// TIA Portal V20 export
// export: Created 2025-12-01T14:57:06.3862051Z, ExportSetting None, DisplayName Totally Integrated Automation Portal, DisplayVersion V20 Update 3, DisplayName TIA Portal Openness, DisplayVersion V20 Update 3, DisplayName TIA Portal Version Control Interface, DisplayVersion V20 Update 3, DisplayName STEP 7 Professional, DisplayVersion V20 Update 3, DisplayName STEP 7 Safety, DisplayVersion V20 Update 2, DisplayName WinCC Basic/Comfort/Advanced, DisplayVersion V20 Update 3, DisplayName WinCC Professional, DisplayVersion V20 Update 3, DisplayName WinCC Unified, DisplayVersion V20 Update 3
FUNCTION "FC978_PosiControl_VarLenze" : Void   // FC978, LAD
{ S7_Optimized_Access := 'FALSE' }
// stored: AutoNumber false, SetENOAutomatically false
   VAR_INPUT
      Estado_CB : "EstadoZona";
      Error_Tx : Bool;
      NodoNoPresente : Bool;
      ByteInicial : Int;
      Velocidad_FR : Int;
      MaxVelocidad_FR : Int;
      EM_Up : Bool;
      EM_Dw : Bool;
      pHsProtusion : Bool;
      SubirManual : Bool;
      BajarManual : Bool;
      Homing : Bool;
      ModoHormingAuto : Bool;
      pHsReferencia : Bool;
      Orden : Bool;
      PosicionOrden : Int;
   END_VAR
   VAR_OUTPUT
      Error_SubjetArea : Word;
      Error_IDArea : Word;
      FinOrden : Bool;
   END_VAR
   VAR_IN_OUT
      PosicionActual : Int;
      ReferenciaOK : Bool;
      ErrorVariador : Bool;
      MemoHomingAuto : Bool;
   END_VAR
   VAR_TEMP
      InVar : Struct
         EnPosicion : Bool;   // Indica que el variador esta posicionado dentro de unos margenes
         EnMovimiento : Bool;   // Indica que el variador esta realizando una orden
         ReferenciaOK : Bool;   // Indica que el variador esta bien referenciado desde la posicion de origen
         HomingDone : Bool;
         SelecMotor_Bit1 : Bool;
         SelecMotor_Bit2 : Bool;
         Libre_Bit14 : Bool;
         Libre_Bit15 : Bool;
         Error_Var : Bool;   // Esto nos indica que hay un erro en el variador
         Libre_Bit1 : Bool;
         Libre_Bit2 : Bool;
         Inhivido : Bool;   // Señal Inhivir var actibo
         Ready_Var : Bool;   // Nos indica que el variador esta listo para realizar los movimientos
         Libre_Bit5 : Bool;
         Libre_Bit6 : Bool;
         Welltime : Bool;
      END_STRUCT;
      OutVar : Struct
         Ejecutar_Posicionamiento : Bool;   // Se activa para dar marcha
         EnableSpeedOveride : Bool;   // Para habilitar el speedoveride
         Reset_Homing : Bool;   // Para referenciar de nuevo el elevador
         Rearme_Var : Bool;
         Set_Homing : Bool;
         pHsReferencia : Bool;
         Manual_Subir : Bool;
         Manual_Bajar : Bool;
         Libre_Bit0 : Bool;
         Libre_Bit1 : Bool;
         Libre_Bit2 : Bool;
         Inhivir_Variador : Bool;   // Señal para inhivir el variador
         Modo_Homming : Bool;   // Tiene que estar activado para refernciar el elevador a cero
         Modo_Manual : Bool;   // Tiene que estar a uno para hacer movimiento en manual
         Modo_AutoRemoto : Bool;   // Tiene que estar a uno para lanzar el posicionamiento
         Libre_Bit7 : Bool;
      END_STRUCT;
      SpeedOrverride : Int;
      P_InVar : DWord;
      P_OutVar : DWord;
      PosicionDestino : Int;
      P_ByteInicialVar : DWord;
      P_Temporal : DWord;
      TempVelocidad : DInt;
      TempVelocidadMax : DInt;
      Margen : Int;
      PosDestinoMinimo : Int;
      PosDestinoMaximo : Int;
   END_VAR
BEGIN

REGION Network 1: Inicializacion
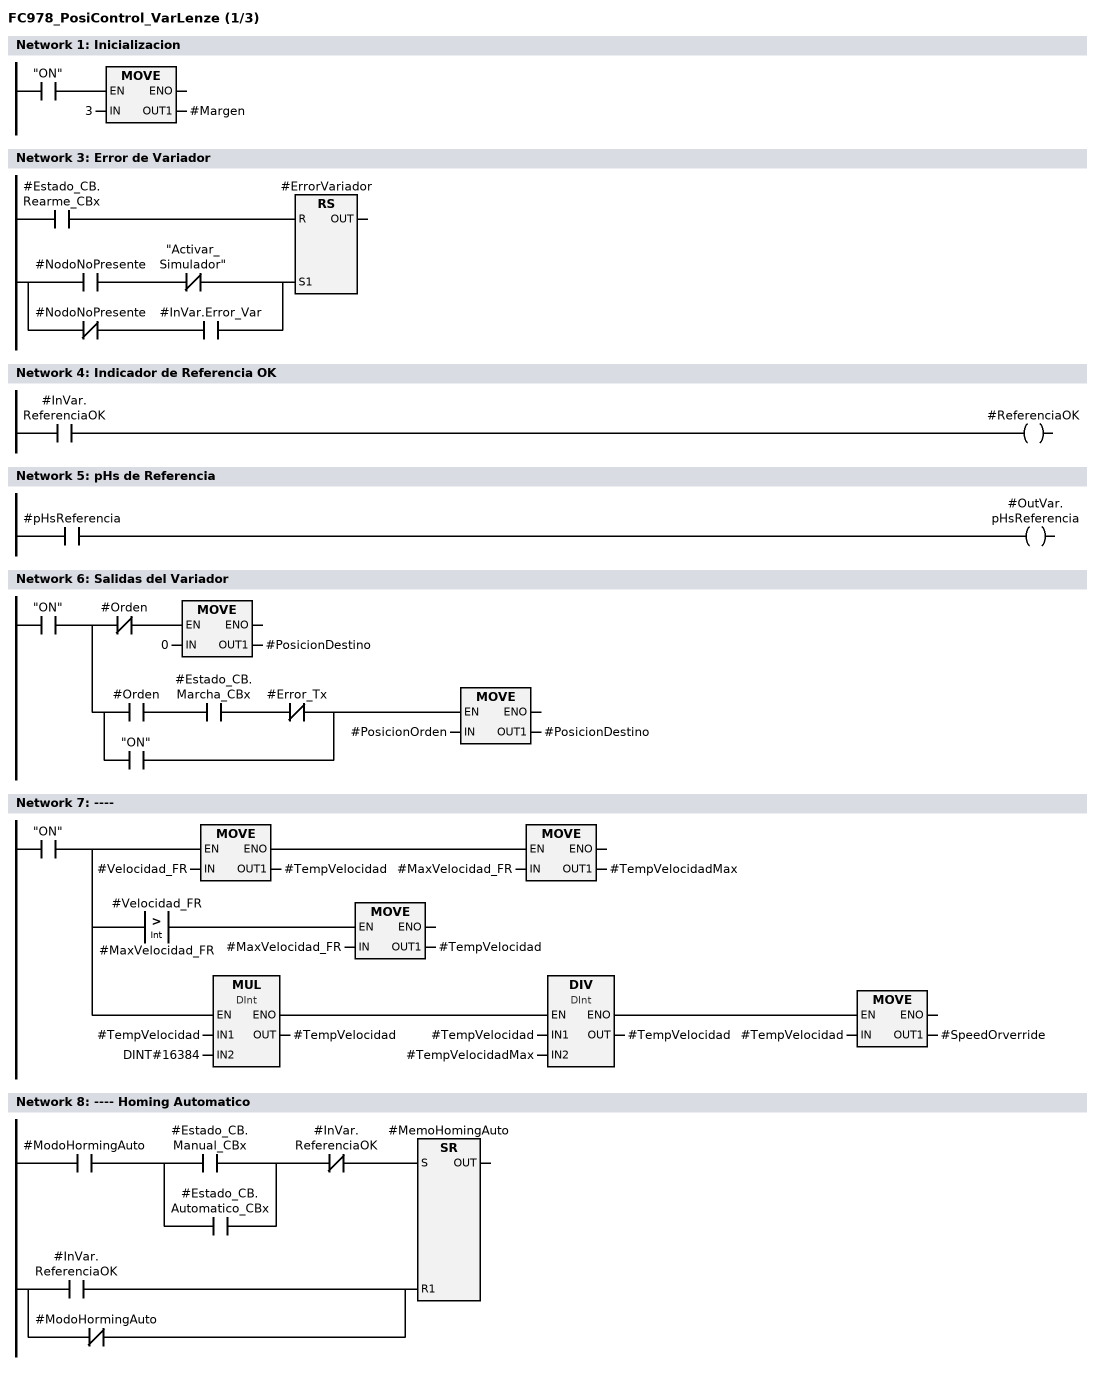
   RUNG wire#powerrail
      Contact( "ON" )
      { S7_GenerateENO := "TRUE" } Move(in := 3, out1 => #Margen)
   END_RUNG
   // the same network as SCL:
   IF "ON" THEN #Margen := 3; END_IF;
END_REGION

NETWORK
TITLE = Lectura del Variador
// -------------------------------------------------------------------
// --- Inicializar las Variables Internas

      L     P##InVar;  // Punteros a las variables internas
      T     #P_InVar;
      L     P##OutVar;
      T     #P_OutVar;

      L     #ByteInicial;  // Puntero al Variador
      SLD   3;
      T     #P_ByteInicialVar;

      L     0;  // Inicializar las variables internas
      T     LW [#P_InVar];
      T     LW [#P_OutVar];

      A     #NodoNoPresente;
      JC    NoLecturaVariador;

// -------------------------------------------------------------------
// --- Lectura de Datos del Variador

      L     #P_ByteInicialVar;  // Leer el Word p#0.0 del Variador
      L     P#0.0;  // Status del Variador "IN"
      +D;
      T     #P_Temporal;

      L     IW [#P_Temporal];
      T     LW [#P_InVar];

      L     #P_ByteInicialVar;  // Leer el Word p#2.0 del Variador
      L     P#2.0;  // Posicion Actual
      +D;
      T     #P_Temporal;

      L     IW [#P_Temporal];
      T     #PosicionActual;

// --- Codigo de Error

      L     #P_ByteInicialVar;  // Leer el Word p#6.0 del Variador
      L     P#6.0;  // ID Area del Variador
      +D;
      T     #P_Temporal;

      L     IW [#P_Temporal];
      T     #Error_IDArea;

      L     #P_ByteInicialVar;  // Leer el Word p#8.0 del Variador
      L     P#8.0;  // Subject Area del Variador
      +D;
      T     #P_Temporal;

      L     IW [#P_Temporal];
      T     #Error_SubjetArea;

// -------------------------------------------------------------------
// --- Final de Lectura de Datos del Variados

NoLecturaVariador:NOP   0;


REGION Network 3: Error de Variador
   RUNG wire#powerrail
      Contact( #Estado_CB.Rearme_CBx )
      S_RS(operand := #ErrorVariador, s1 := wire#w1)
   END_RUNG
   RUNG wire#powerrail
      Contact( #NodoNoPresente )
      I_Contact( "Activar_Simulador" )
   END_RUNG wire#w1
   RUNG wire#powerrail
      I_Contact( #NodoNoPresente )
      Contact( #InVar.Error_Var )
   END_RUNG wire#w1
   // the same network as SCL:
   IF #Estado_CB.Rearme_CBx THEN
       #ErrorVariador := FALSE;   // RS flip-flop
   END_IF;
   IF (#NodoNoPresente AND NOT "Activar_Simulador") OR (NOT #NodoNoPresente AND #InVar.Error_Var) THEN
       #ErrorVariador := TRUE;
   END_IF;
END_REGION

REGION Network 4: Indicador de Referencia OK
   RUNG wire#powerrail
      Contact( #InVar.ReferenciaOK )
      Coil( #ReferenciaOK )
   END_RUNG
   // the same network as SCL:
   #ReferenciaOK := #InVar.ReferenciaOK;
END_REGION

REGION Network 5: pHs de Referencia
   RUNG wire#powerrail
      Contact( #pHsReferencia )
      Coil( #OutVar.pHsReferencia )
   END_RUNG
   // the same network as SCL:
   #OutVar.pHsReferencia := #pHsReferencia;
END_REGION

REGION Network 6: Salidas del Variador
   RUNG wire#powerrail
      Contact( "ON" )
      wire#w1
      I_Contact( #Orden )
      { S7_GenerateENO := "TRUE" } Move(in := 0, out1 => #PosicionDestino)
   END_RUNG
   RUNG wire#w1
      Contact( #Orden )
      Contact( #Estado_CB.Marcha_CBx )
      I_Contact( #Error_Tx )
      wire#w2
      { S7_GenerateENO := "TRUE" } Move(in := #PosicionOrden, out1 => #PosicionDestino)
   END_RUNG
   RUNG wire#w1
      Contact( "ON" )
   END_RUNG wire#w2
   // the same network as SCL:
   IF "ON" AND NOT #Orden THEN #PosicionDestino := 0; END_IF;
   IF "ON" AND ((#Orden AND #Estado_CB.Marcha_CBx AND NOT #Error_Tx) OR "ON") THEN
       #PosicionDestino := #PosicionOrden;
   END_IF;
END_REGION

REGION Network 7: ----
   RUNG wire#powerrail
      Contact( "ON" )
      wire#w1
      { S7_GenerateENO := "TRUE" } Move(in := #Velocidad_FR, out1 => #TempVelocidad)
      { S7_GenerateENO := "TRUE" } Move(in := #MaxVelocidad_FR, out1 => #TempVelocidadMax)
   END_RUNG
   RUNG wire#w1
      { S7_Templates := "SrcType := Int" } GT_Contact(in1 := #Velocidad_FR, in2 := #MaxVelocidad_FR)
      { S7_GenerateENO := "TRUE" } Move(in := #MaxVelocidad_FR, out1 => #TempVelocidad)
   END_RUNG
   RUNG wire#w1
      { S7_Templates := "SrcType := DInt"; S7_GenerateENO := "TRUE" } Mul(in1 := #TempVelocidad, in2 := DINT#16384, out => #TempVelocidad)
      { S7_Templates := "SrcType := DInt"; S7_GenerateENO := "TRUE" } Div(in1 := #TempVelocidad, in2 := #TempVelocidadMax, out => #TempVelocidad)
      { S7_GenerateENO := "TRUE" } Move(in := #TempVelocidad, out1 => #SpeedOrverride)
   END_RUNG
   // the same network as SCL:
   // ENO of a box is taken as its EN; it also drops when the box reports an error
   IF "ON" THEN
       #TempVelocidad := #Velocidad_FR;
       #TempVelocidadMax := #MaxVelocidad_FR;
   END_IF;
   IF "ON" AND (#Velocidad_FR > #MaxVelocidad_FR) THEN #TempVelocidad := #MaxVelocidad_FR; END_IF;
   IF "ON" THEN
       #TempVelocidad := #TempVelocidad * DINT#16384;
       #TempVelocidad := #TempVelocidad / #TempVelocidadMax;
       #SpeedOrverride := #TempVelocidad;
   END_IF;
END_REGION

REGION Network 8: ---- Homing Automatico
   RUNG wire#powerrail
      Contact( #ModoHormingAuto )
      wire#w1
      Contact( #Estado_CB.Manual_CBx )
      wire#w2
      I_Contact( #InVar.ReferenciaOK )
      S_SR(operand := #MemoHomingAuto, r1 := wire#w3)
   END_RUNG
   RUNG wire#w1
      Contact( #Estado_CB.Automatico_CBx )
   END_RUNG wire#w2
   RUNG wire#powerrail
      Contact( #InVar.ReferenciaOK )
   END_RUNG wire#w3
   RUNG wire#powerrail
      I_Contact( #ModoHormingAuto )
   END_RUNG wire#w3
   // the same network as SCL:
   IF #ModoHormingAuto AND (#Estado_CB.Manual_CBx OR #Estado_CB.Automatico_CBx) AND NOT #InVar.ReferenciaOK THEN
       #MemoHomingAuto := TRUE;   // SR flip-flop
   END_IF;
   IF #InVar.ReferenciaOK OR NOT #ModoHormingAuto THEN #MemoHomingAuto := FALSE; END_IF;
END_REGION

REGION Network 9: ---
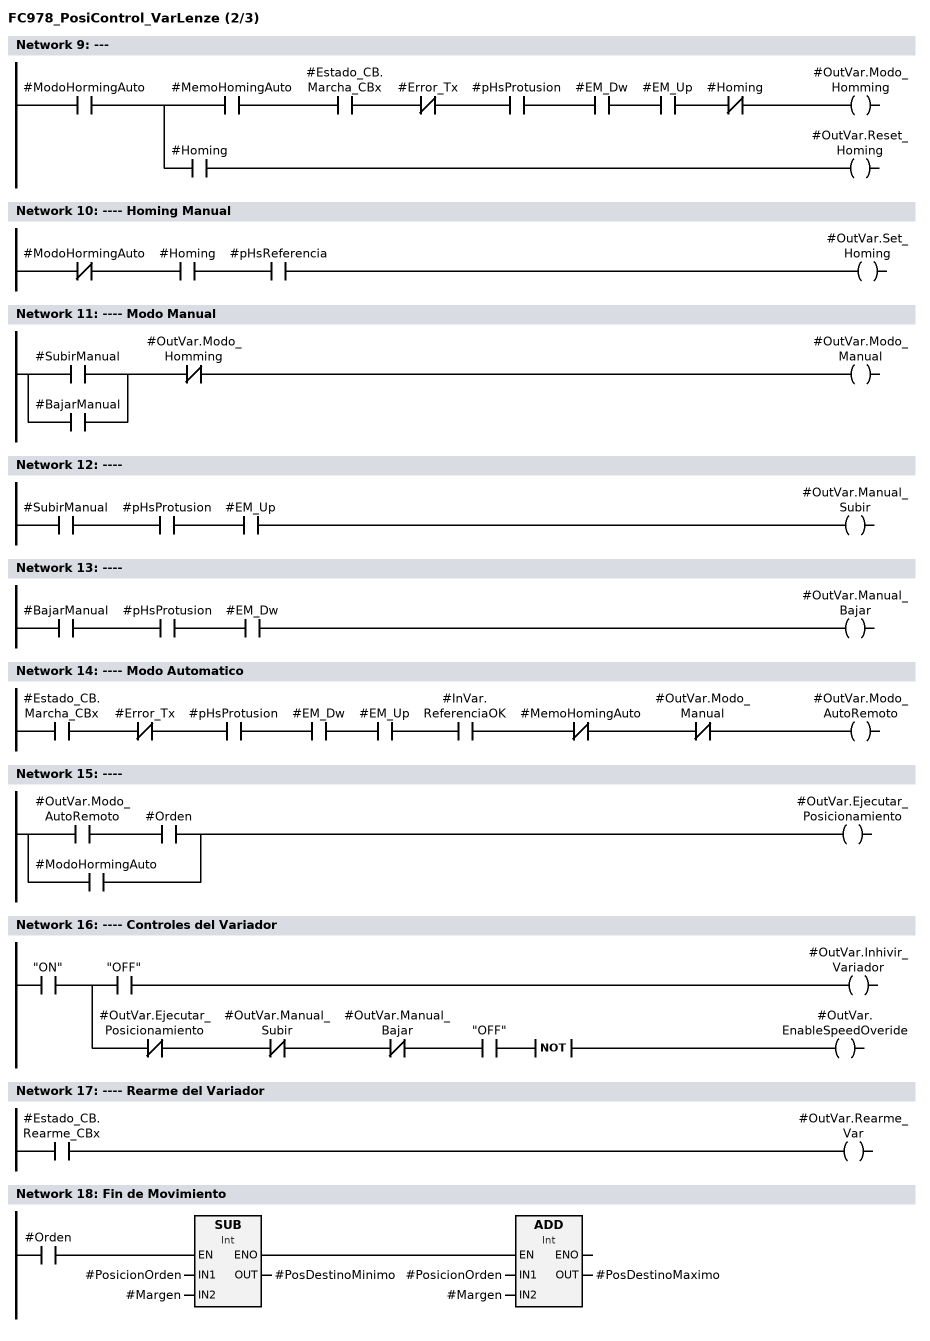
   RUNG wire#powerrail
      Contact( #ModoHormingAuto )
      wire#w1
      Contact( #MemoHomingAuto )
      Contact( #Estado_CB.Marcha_CBx )
      I_Contact( #Error_Tx )
      Contact( #pHsProtusion )
      Contact( #EM_Dw )
      Contact( #EM_Up )
      I_Contact( #Homing )
      Coil( #OutVar.Modo_Homming )
   END_RUNG
   RUNG wire#w1
      Contact( #Homing )
      Coil( #OutVar.Reset_Homing )
   END_RUNG
   // the same network as SCL:
   #OutVar.Modo_Homming := #ModoHormingAuto AND #MemoHomingAuto AND #Estado_CB.Marcha_CBx AND NOT #Error_Tx AND #pHsProtusion AND #EM_Dw AND #EM_Up AND NOT #Homing;
   #OutVar.Reset_Homing := #ModoHormingAuto AND #Homing;
END_REGION

REGION Network 10: ---- Homing Manual
   RUNG wire#powerrail
      I_Contact( #ModoHormingAuto )
      Contact( #Homing )
      Contact( #pHsReferencia )
      Coil( #OutVar.Set_Homing )
   END_RUNG
   // the same network as SCL:
   #OutVar.Set_Homing := NOT #ModoHormingAuto AND #Homing AND #pHsReferencia;
END_REGION

REGION Network 11: ---- Modo Manual
   RUNG wire#powerrail
      Contact( #SubirManual )
      wire#w1
      I_Contact( #OutVar.Modo_Homming )
      Coil( #OutVar.Modo_Manual )
   END_RUNG
   RUNG wire#powerrail
      Contact( #BajarManual )
   END_RUNG wire#w1
   // the same network as SCL:
   #OutVar.Modo_Manual := (#SubirManual OR #BajarManual) AND NOT #OutVar.Modo_Homming;
END_REGION

REGION Network 12: ----
   RUNG wire#powerrail
      Contact( #SubirManual )
      Contact( #pHsProtusion )
      Contact( #EM_Up )
      Coil( #OutVar.Manual_Subir )
   END_RUNG
   // the same network as SCL:
   #OutVar.Manual_Subir := #SubirManual AND #pHsProtusion AND #EM_Up;
END_REGION

REGION Network 13: ----
   RUNG wire#powerrail
      Contact( #BajarManual )
      Contact( #pHsProtusion )
      Contact( #EM_Dw )
      Coil( #OutVar.Manual_Bajar )
   END_RUNG
   // the same network as SCL:
   #OutVar.Manual_Bajar := #BajarManual AND #pHsProtusion AND #EM_Dw;
END_REGION

REGION Network 14: ---- Modo Automatico
   RUNG wire#powerrail
      Contact( #Estado_CB.Marcha_CBx )
      I_Contact( #Error_Tx )
      Contact( #pHsProtusion )
      Contact( #EM_Dw )
      Contact( #EM_Up )
      Contact( #InVar.ReferenciaOK )
      I_Contact( #MemoHomingAuto )
      I_Contact( #OutVar.Modo_Manual )
      Coil( #OutVar.Modo_AutoRemoto )
   END_RUNG
   // the same network as SCL:
   #OutVar.Modo_AutoRemoto := #Estado_CB.Marcha_CBx AND NOT #Error_Tx AND #pHsProtusion AND #EM_Dw AND #EM_Up AND #InVar.ReferenciaOK AND NOT #MemoHomingAuto AND NOT #OutVar.Modo_Manual;
END_REGION

REGION Network 15: ----
   RUNG wire#powerrail
      Contact( #OutVar.Modo_AutoRemoto )
      Contact( #Orden )
      wire#w1
      Coil( #OutVar.Ejecutar_Posicionamiento )
   END_RUNG
   RUNG wire#powerrail
      Contact( #ModoHormingAuto )
   END_RUNG wire#w1
   // the same network as SCL:
   #OutVar.Ejecutar_Posicionamiento := (#OutVar.Modo_AutoRemoto AND #Orden) OR #ModoHormingAuto;
END_REGION

REGION Network 16: ---- Controles del Variador
   RUNG wire#powerrail
      Contact( "ON" )
      wire#w1
      Contact( "OFF" )
      Coil( #OutVar.Inhivir_Variador )
   END_RUNG
   RUNG wire#w1
      I_Contact( #OutVar.Ejecutar_Posicionamiento )
      I_Contact( #OutVar.Manual_Subir )
      I_Contact( #OutVar.Manual_Bajar )
      Contact( "OFF" )
      Not()
      Coil( #OutVar.EnableSpeedOveride )
   END_RUNG
   // the same network as SCL:
   #OutVar.Inhivir_Variador := "ON" AND "OFF";
   #OutVar.EnableSpeedOveride := NOT ("ON" AND NOT #OutVar.Ejecutar_Posicionamiento AND NOT #OutVar.Manual_Subir AND NOT #OutVar.Manual_Bajar AND "OFF");
END_REGION

REGION Network 17: ---- Rearme del Variador
   RUNG wire#powerrail
      Contact( #Estado_CB.Rearme_CBx )
      Coil( #OutVar.Rearme_Var )
   END_RUNG
   // the same network as SCL:
   #OutVar.Rearme_Var := #Estado_CB.Rearme_CBx;
END_REGION

REGION Network 18: Fin de Movimiento
   RUNG wire#powerrail
      Contact( #Orden )
      { S7_Templates := "SrcType := Int"; S7_GenerateENO := "TRUE" } Sub(in1 := #PosicionOrden, in2 := #Margen, out => #PosDestinoMinimo)
      { S7_Templates := "SrcType := Int"; S7_GenerateENO := "TRUE" } Add(in1 := #PosicionOrden, in2 := #Margen, out => #PosDestinoMaximo)
   END_RUNG
   // the same network as SCL:
   // ENO of a box is taken as its EN; it also drops when the box reports an error
   IF #Orden THEN
       #PosDestinoMinimo := #PosicionOrden - #Margen;
       #PosDestinoMaximo := #PosicionOrden + #Margen;
   END_IF;
END_REGION

REGION Network 19: ----
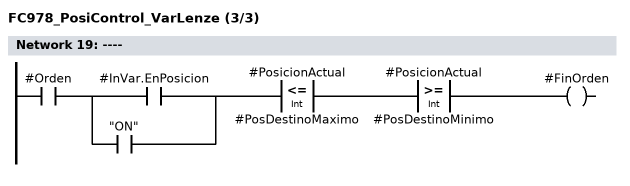
   RUNG wire#powerrail
      Contact( #Orden )
      wire#w1
      Contact( #InVar.EnPosicion )
      wire#w2
      { S7_Templates := "SrcType := Int" } LE_Contact(in1 := #PosicionActual, in2 := #PosDestinoMaximo)
      { S7_Templates := "SrcType := Int" } GE_Contact(in1 := #PosicionActual, in2 := #PosDestinoMinimo)
      Coil( #FinOrden )
   END_RUNG
   RUNG wire#w1
      Contact( "ON" )
   END_RUNG wire#w2
   // the same network as SCL:
   #FinOrden := #Orden AND (#InVar.EnPosicion OR "ON") AND (#PosicionActual <= #PosDestinoMaximo) AND (#PosicionActual >= #PosDestinoMinimo);
END_REGION

NETWORK
TITLE = Escritura del Variador

      A     #NodoNoPresente;
      JC    NoEscrituraVariador;

// -------------------------------------------------------------------
// --- Escritura de Datos del Variador

      L     #P_ByteInicialVar;  // Escritura el Word p#4.0 del Variador
      L     P#4.0;  // Posicion a Moverse
      +D;
      T     #P_Temporal;

      L     #PosicionDestino;
      T     QW [#P_Temporal];

      L     #P_ByteInicialVar;  // Escritura el Word p#0.0 del Variador
      L     P#0.0;  // Status del Variador "OUT"
      +D;
      T     #P_Temporal;

      L     LW [#P_OutVar];
      T     QW [#P_Temporal];

      L     #P_ByteInicialVar;  // Escritura el Word p#2.0 del Variador
      L     P#2.0;  // Velocidad de Movimiento
      +D;
      T     #P_Temporal;

      L     #SpeedOrverride;
      T     QW [#P_Temporal];

// -------------------------------------------------------------------
// --- Final de Escritura de Datos del Variados

NoEscrituraVariador:NOP   0;


END_FUNCTION
